{attribute 'linkalways'} 
{attribute 'no_explicit_call' := 'This FB is a CLASS and must be accessed using methods or properties'}
{attribute 'enable_dynamic_creation'}
FUNCTION_BLOCK _TcVnVector4_UINT EXTENDS AliasDatatypeBase
VAR
	localData : TcVnVector4_UINT;
	activeData : REFERENCE TO TcVnVector4_UINT REF= localData;
	aliasBaseDatatype : _Array0to3OfUINT;
END_VAR

PROPERTY PUBLIC Address : PVOID
GET
Address := ADR(activeData);
END_GET
END_PROPERTY

METHOD PUBLIC ClearReference
VAR_INPUT
END_VAR
activeData REF= localData;
SetBaseDatatypeReference();
END_METHOD

METHOD PUBLIC Clone : I_Datatype
VAR
    pClone : POINTER TO _TcVnVector4_UINT;
END_VAR
pClone := __NEW(_TcVnVector4_UINT);
Clone := pClone^;
END_METHOD

METHOD FB_init : BOOL
VAR_INPUT
	bInitRetains : BOOL; // if TRUE, the retain variables are initialized (warm start / cold start)
	bInCopyCode : BOOL;  // if TRUE, the instance afterwards gets moved into the copy code (online change)
	//InitialValue : <type>; // if possible, not all values can be initialized
END_VAR
//localData := InitialValue; // if possible, not all values can be initialized
SetBaseDatatypeReference();
AddBaseDatatype(aliasBaseDatatype);
END_METHOD

PROPERTY PUBLIC Identifier : T_MAXSTRING
GET
Identifier := 'TcVnVector4_UINT';
END_GET
END_PROPERTY

METHOD PUBLIC MakeReferenceTo
VAR_INPUT
	ReferenceTarget : REFERENCE TO TcVnVector4_UINT;
END_VAR
activeData REF= ReferenceTarget;
SetBaseDatatypeReference();
END_METHOD

METHOD PROTECTED SetBaseDatatypeReference
VAR_INPUT
END_VAR
aliasBaseDatatype.MakeReferenceTo(activeData);
END_METHOD

PROPERTY PUBLIC Size : UDINT
GET
Size := SIZEOF(activeData);
END_GET
END_PROPERTY

METHOD TryMakeReferenceTo : BOOL
VAR_INPUT
	Target : I_Datatype;
END_VAR
VAR
	targetAsAlias : I_AliasDatatype;
	pTargetData : POINTER TO TcVnVector4_UINT;
END_VAR
IF NOT Target.TryResolveAsAliasDatatype(targetAsAlias) THEN
	RETURN;
END_IF

IF targetAsAlias.Identifier <> Identifier THEN
	RETURN;
END_IF

pTargetData := Target.Address;
activeData REF= pTargetData^;
SetBaseDatatypeReference();
TryMakeReferenceTo := TRUE;
END_METHOD

PROPERTY PUBLIC Value : REFERENCE TO TcVnVector4_UINT
GET
Value REF= activeData;
END_GET
END_PROPERTY

END_FUNCTION_BLOCK

(* stored: Version 1.1.0.1, ProductVersion 3.1.4024.13
   POU _TcVnVector4_UINT: Id {50b3538e-35bc-0e22-0379-865c2096ffb2}, SpecialFunc None
   Folder Core: Id {ac5caff0-8e3c-08da-0ec5-2fdb8d1ec564}
   Folder Protected: Id {f92ec475-2dc7-0d8b-26ea-41574a3eecfc}
   Folder Customize: Id {1083e6c2-2e8c-0ab6-02bb-beef58a444a4}
   Folder Constructor: Id {23607d94-34c7-04df-0b34-b4f3fb6d1739}
   Property Address: Id {5914826d-477b-04ad-2b8a-2252dd6d3da6}
   Get Get: Id {54d8d09d-31fc-02c5-3609-51bb9677981c}
   Method ClearReference: Id {afb49732-56b1-01a3-0429-360331e0e146}
   Method Clone: Id {04eeaa75-ebbe-0fab-220f-a6c7c749a0f1}
   Method FB_init: Id {b9032d92-70be-0543-2980-f6629a36b939}
   Property Identifier: Id {66797fb5-743d-09a3-1a6d-da5bbede0739}
   Get Get: Id {693f6679-5d3e-0ca6-2bf4-981b01ab7166}
   Method MakeReferenceTo: Id {14b34e43-5666-09e2-1a1d-4066371cfeda}
   Method SetBaseDatatypeReference: Id {165f2f1a-a213-0dd9-2c7c-59f83ddfc050}
   Property Size: Id {a17a2e46-389e-0f64-2009-28d159cc53eb}
   Get Get: Id {287463bf-b64a-0e50-1268-beb839e91c7e}
   Method TryMakeReferenceTo: Id {f7d8700b-cced-034f-1a56-71a082add33a}
   Property Value: Id {0c0cea34-2784-08a7-3434-279d7cfc8e28}
   Get Get: Id {133bfaab-0f19-00a1-0278-bb6ab0abe169} *)
